TYPE ST_PitchControl :
STRUCT
	Enable: BOOL;
	Reset: BOOL;
	ReduceTorque: BOOL;
	Velocity: INT;
END_STRUCT
END_TYPE

(* stored: Version 1.1.0.1, ProductVersion 3.1.4026.18
   DUT ST_PitchControl: Id {7019d56a-699f-4bcd-8d6a-2cbfa712afee} *)
